IF NOT (Transfer.Mode = FIT_VFD_Transfer_Modes.Pause) AND NOT (Transfer.Mode = FIT_VFD_Transfer_Modes.Resume) THEN _w1 := Transfer.Mode; END_IF
Transfer.Config.Mode_Memory := _w1;
IF Transfer.Mode = FIT_VFD_Transfer_Modes.Resume THEN _w2 := Transfer.Config.Mode_Memory; END_IF
Transfer.Mode := _w2;
Transfer.Status := SEL(False, SEL(BCV_Not_Ready, SEL(ACV_Not_Ready, SEL(Transfer.Mode=FIT_VFD_Transfer_Modes.Lock_Out, SEL(False, SEL(Complete, SEL(Transfer_Running, SEL(FIT.PLC_Reset, SEL(IDLE_Return, SEL(PAUSED, Transfer_status.IDLE, Transfer_status.Paused), Transfer_status.IDLE), Transfer_status.FIT_Reset), Transfer_status.Running), Transfer_status.Complete), Transfer_status.Complete), Transfer_status.LOCKED_OUT), Transfer_status.ACV_Not_Ready), Transfer_status.BCV_Not_Ready), Transfer_status.VFD_Not_Ready);
_w3 := Transfer.Mode = FIT_VFD_Transfer_Modes.Idle;
_w4 := True AND NOT (ACV.Mode = ACV_Modes.Auto);
ACV_Not_Ready := _w3 AND _w4;
_w5 := _w4 OR False;
SR2(SET1 := _w3 AND _w5, RESET := NOT _w5); // SR
IF SR2.Q1 THEN _w6 := FIT_VFD_Transfer_Modes.Idle; END_IF
Transfer.Mode := _w6;
_w7 := Transfer.Status = Transfer_Status.Complete;
_w8 := Transfer_Status.IDLE = Transfer.Status OR False OR Transfer.Status = Transfer_Status.LOCKED_OUT;
_w9 := Transfer.Status = Transfer_Status.BCV_Not_Ready;
_w10 := Transfer.Mode = FIT_VFD_Transfer_Modes.Pause;
PAUSED := _w10;
_w11 := Transfer.Mode = FIT_VFD_Transfer_Modes.IDLE;
_w12 := Complete OR Error OR _w11 OR _w10;
CTRL_PID_1(
    ACT := FIT.Rate,
    SET := Transfer.Config.Target_Rate,
    SUP := 0.0,
    OFS := Transfer.Config.Target_Rate * Transfer.Config.FF,
    M_I := 0.0,
    MAN := _w12,
    RST := _w12,
    KP := Transfer.Config.KP,
    TN := Transfer.Config.TN,
    TV := Transfer.Config.TV,
    LL := 0,
    LH := 100); // BURKERT_OSCAT_BASIC.CTRL_PID
PID_CV := CTRL_PID_1.Y;
TP11(IN := NOT LockOut_Active AND _w12, PT := t#2s); // TP
ACV.PLC_CMD := SEL(TP11.Q, ACV.PLC_CMD, 0.0);
IDLE_Return := _w9 AND _w11;
SR_10(SET1 := FIT.Total<1, RESET := _w11); // SR
TON_10(IN := SR_10.Q1, PT := T#2s); // TON
FIT_Reset_Complete := TON_10.Q;
R_TRIG_0(CLK := _w11 OR TON_10.Q); // R_trig
_w13 := SEL(R_TRIG_0.Q, FIT.PLC_Reset, False);
_w14 := Transfer.Mode = FIT_VFD_Transfer_Modes.Batch;
_w15 := _w14 AND FIT_Reset_Complete AND FIT.Total >= Transfer.Config.Target_Volume;
Batch_Complete := _w15;
RS_11(SET := Time_Complete OR _w15 OR False, RESET1 := _w11); // RS
Complete := RS_11.Q1;
_w16 := LOCK_OUT AND _w8 AND NOT RS_11.Q1;
F_TRIG_10(CLK := _w16); // F_Trig
IF F_TRIG_10.Q THEN _w17 := FIT_VFD_Transfer_Modes.Idle; END_IF
Transfer.Mode := _w17;
_w18 := _w16;
IF _w18 THEN _w19 := FIT_VFD_Transfer_Modes.Lock_Out; END_IF
LockOut_Active := _w18;
Transfer.Mode := _w19;
FIT.PLC_Reset := SEL(NOT SR_10.Q1 AND _w14 AND NOT _w15, _w13, True);
_w20 := _w14 AND FIT_Reset_Complete AND NOT Complete AND NOT Error AND NOT Time_Complete;
Transfer_Running := _w20;
transfer.Remaining_Volume := SEL(_w20, Transfer.Config.Target_Volume, Transfer.Config.Target_Volume-fit.Total);
ACV.PLC_CMD := SEL(_w20, ACV.PLC_CMD, PID_CV);
TON_12(IN := _w7, PT := T#10s); // TON

END_FUNCTION_BLOCK

// 20 Program Organization Units/Level_2_Controls/Batch
FUNCTION_BLOCK Batch
VAR_INPUT
	Rate_PID: REFERENCE TO PID_Control;
	Config:	REFERENCE TO cBatch;
	FIT_Total:REAL;
	FIT_Rate:REAL;
	
END_VAR
VAR_OUTPUT
	FIT_Reset:BOOL;
END_VAR
VAR
	Local_Status:eBatch_Status;
	Local_task:eBatch_Task;
	Local_mode:eHOA_Modes;
	
	Start_Rate:REAL;
	End_Rate:REAL;
	
END_VAR

//AUX(); Now Called From Methods


CASE Config.Line_Mode.eMode OF
	eHOA_Modes.Auto:Mode_Auto();
	eHOA_Modes.Manual:Mode_Manual();
	eHOA_Modes.Off:Mode_OFF();
	
END_CASE;

CASE Config.Line_Task.eTask OF
	eBatch_Task.OFF:Task_off();
	eBAtch_Task.Pause:Task_Pause();
	eBatch_Task.Resume:Task_Resume();
	eBatch_task.Run:Task_Run();
	
END_CASE

END_FUNCTION_BLOCK

// 20 Program Organization Units/Transfer_ACV_VFD_FIT_UDFB
FUNCTION_BLOCK Transfer_ACV_VFD_FIT_UDFB
VAR_INPUT
	//Index:INT;
	LOCK_OUT:BOOL:=FALSE;
	
END_VAR
VAR_OUTPUT
END_VAR
VAR
	Paused:BOOL;
	Idle_return:BOOL;
	Transfer_Running:BOOL;
	Complete:BOOL;
	ACV_Not_Ready:BOOL;
	VFD_Not_Ready:BOOL;
	BCV_Not_Ready:BOOL;
	Time_Complete:BOOL;
	FIT_Reset_Complete:BOOL;
	Pump_Start:BOOL;
	Lockout_Active:BOOL;
	Error:BOOL;
	Flow_Mode:BOOL;
	Batch_Complete:BOOL;
	Enable_pump:BOOL;
	
	PID_CV:REAL;
	
	
	
	
	SR2: SR;
	TON_0: TON;
	CTRL_PID_1: BURKERT_OSCAT_BASIC.CTRL_PID;
	R_TRIG_0: R_trig;
	TON_10: TON;
	SR_10: SR;
	RS_11: RS;
	TON_12: TON;
	F_TRIG_10: F_Trig;
	TP11: TP;
END_VAR

VAR_IN_OUT
	Transfer:FIT_VFD_Transfer_DUT;
	VFD:VFD_Vacon_DUT;
	ACV:ACV_DUT;
	FIT:FIT_DUT;
	
END_VAR
VAR // added by the converter: edge detectors and wires of the graphical bodies
    _w1, _w2, _w7, _w22, _w24 : ANY;
    _w3, _w4, _w5, _w6, _w8, _w9, _w10, _w11, _w12, _w13, _w14, _w15, _w16, _w17, _w18, _w19, _w20, _w21, _w23, _w25 : BOOL;
END_VAR

IF NOT (Transfer.Mode = FIT_VFD_Transfer_Modes.Pause) AND NOT (Transfer.Mode = FIT_VFD_Transfer_Modes.Resume) THEN _w1 := Transfer.Mode; END_IF
Transfer.Config.Mode_Memory := _w1;
IF Transfer.Mode = FIT_VFD_Transfer_Modes.Resume THEN _w2 := Transfer.Config.Mode_Memory; END_IF
Transfer.Mode := _w2;
Transfer.Status := SEL(VFD_Not_Ready, SEL(BCV_Not_Ready, SEL(ACV_Not_Ready, SEL(Transfer.Mode=FIT_VFD_Transfer_Modes.Lock_Out, SEL(False, SEL(Complete, SEL(Transfer_Running, SEL(FIT.PLC_Reset, SEL(IDLE_Return, SEL(PAUSED, Transfer_status.IDLE, Transfer_status.Paused), Transfer_status.IDLE), Transfer_status.FIT_Reset), Transfer_status.Running), Transfer_status.Complete), Transfer_status.Complete), Transfer_status.LOCKED_OUT), Transfer_status.ACV_Not_Ready), Transfer_status.BCV_Not_Ready), Transfer_status.VFD_Not_Ready);
_w3 := Transfer.Mode = FIT_VFD_Transfer_Modes.Idle;
_w4 := True AND NOT (ACV.Mode = ACV_Modes.Auto);
ACV_Not_Ready := _w3 AND _w4;
_w5 := True AND NOT (VFD.CONTROL.MODE = VFD_Modes.Auto);
_w6 := _w4 OR _w5;
SR2(SET1 := _w3 AND _w6, RESET := NOT _w6); // SR
IF SR2.Q1 THEN _w7 := FIT_VFD_Transfer_Modes.Idle; END_IF
Transfer.Mode := _w7;
VFD_Not_Ready := _w3 AND _w5;
_w8 := Transfer.Status = Transfer_Status.Complete;
_w9 := Transfer.Status = Transfer_Status.BCV_Not_Ready OR Transfer.Status = Transfer_Status.VFD_Not_Ready;
_w10 := Transfer_Status.IDLE = Transfer.Status OR False OR Transfer.Status = Transfer_Status.LOCKED_OUT;
_w11 := Transfer.Mode = FIT_VFD_Transfer_Modes.Pause;
PAUSED := _w11;
_w12 := Transfer.Mode = FIT_VFD_Transfer_Modes.IDLE;
_w13 := Complete OR Error OR _w12 OR _w11;
_w14 := NOT Pump_Start OR _w13;
CTRL_PID_1(
    ACT := FIT.Rate,
    SET := Transfer.Config.Target_Rate,
    SUP := 0.0,
    OFS := Transfer.Config.Target_Rate * Transfer.Config.FF,
    M_I := 0.0,
    MAN := _w14,
    RST := _w14,
    KP := Transfer.Config.KP,
    TN := Transfer.Config.TN,
    TV := Transfer.Config.TV,
    LL := 0,
    LH := 100); // BURKERT_OSCAT_BASIC.CTRL_PID
PID_CV := CTRL_PID_1.Y;
TP11(IN := NOT LockOut_Active AND _w13, PT := t#2s); // TP
VFD.CONTROL.PLC_Run := SEL(TP11.Q, VFD.CONTROL.PLC_Run, FALSE);
VFD.CONTROL.PLC_CMD := SEL(TP11.Q, VFD.CONTROL.PLC_CMD, 0.0);
ACV.PLC_CMD := SEL(TP11.Q, ACV.PLC_CMD, 0.0);
IDLE_Return := _w9 AND _w12;
SR_10(SET1 := FIT.Total<1, RESET := _w12); // SR
TON_10(IN := SR_10.Q1, PT := T#2s); // TON
FIT_Reset_Complete := TON_10.Q;
R_TRIG_0(CLK := _w12 OR TON_10.Q); // R_trig
_w15 := SEL(R_TRIG_0.Q, FIT.PLC_Reset, False);
_w16 := Transfer.Mode = FIT_VFD_Transfer_Modes.Batch;
_w17 := False OR False OR _w16;
Flow_Mode := _w17;
_w18 := _w17 AND FIT_Reset_Complete AND NOT Complete AND NOT Error AND NOT Time_Complete;
Transfer_Running := _w18;
transfer.Remaining_Volume := SEL(_w18, Transfer.Config.Target_Volume, Transfer.Config.Target_Volume-fit.Total);
_w19 := True AND _w18;
Enable_Pump := _w19;
ACV.PLC_CMD := SEL(_w19, ACV.PLC_CMD, PID_CV);
_w20 := _w16 AND FIT_Reset_Complete AND FIT.Total >= Transfer.Config.Target_Volume;
Batch_Complete := _w20;
RS_11(SET := Time_Complete OR _w20 OR False, RESET1 := _w12); // RS
Complete := RS_11.Q1;
_w21 := LOCK_OUT AND _w10 AND NOT RS_11.Q1;
F_TRIG_10(CLK := _w21); // F_Trig
IF F_TRIG_10.Q THEN _w22 := FIT_VFD_Transfer_Modes.Idle; END_IF
Transfer.Mode := _w22;
_w23 := _w21;
IF _w23 THEN _w24 := FIT_VFD_Transfer_Modes.Lock_Out; END_IF
LockOut_Active := _w23;
Transfer.Mode := _w24;
FIT.PLC_Reset := SEL(NOT SR_10.Q1 AND _w17 AND NOT _w20, _w15, True);
_w25 := SEL(_w19, _w18, ACV.Valve_Actual >= 5);
Pump_Start := _w25;
VFD.CONTROL.PLC_CMD := SEL(_w25, VFD.CONTROL.PLC_CMD, PID_CV);
VFD.CONTROL.PLC_Run := SEL(_w25, VFD.CONTROL.PLC_Run, PID_CV > 15);
TON_12(IN := _w8, PT := T#10s); // TON

END_FUNCTION_BLOCK

// 20 Program Organization Units/Transfer_BCV_FIT_UDFB
FUNCTION_BLOCK Transfer_BCV_FIT_UDFB
VAR_INPUT
	LOCK_OUT:BOOL:=FALSE;
	//FIT_Rate:REAL;
	//FIT_Volume:REAL;
	//Valve_Ready:BOOL;
	
END_VAR
VAR_OUTPUT
	//BCV:BOOL;
	//ACV:REAL:
END_VAR
VAR
	Paused:BOOL;
	Idle_return:BOOL;
	Transfer_Running:BOOL;
	Complete:BOOL;
	ACV_Not_Ready:BOOL;
	//VFD_Not_Ready:BOOL;
	BCV_Not_Ready:BOOL;
	Time_Complete:BOOL;
	FIT_Reset_Complete:BOOL;
	//Pump_Start:BOOL;
	Lockout_Active:BOOL;
	Error:BOOL;
	Flow_Mode:BOOL;
	Batch_Complete:BOOL;
	Enable_pump:BOOL;
	
	//PID_CV:REAL;
	
	
	
	
	SR2: SR;
	TON_0: TON;
	CTRL_PID_1: BURKERT_OSCAT_BASIC.CTRL_PID;
	R_TRIG_0: R_trig;
	TON_10: TON;
	SR_10: SR;
	RS_11: RS;
	TON_12: TON;
	F_TRIG_10: F_Trig;
	TP11: TP;
	FT_PIDW_1: BURKERT_OSCAT_BASIC.FT_PIDW;
	F_TRIG_0: F_Trig;
END_VAR

VAR_IN_OUT
	Transfer:FIT_Transfer_DUT;
	//FIT_Reset:BOOL;
	//VFD:VFD_Vacon_DUT;
	BCV:BCV_DUT;
	FIT:FIT_DUT;
	
END_VAR
VAR // added by the converter: edge detectors and wires of the graphical bodies
    _w1, _w2, _w5, _w6, _w20, _w22, _w23 : ANY;
    _w3, _w4, _w7, _w8, _w9, _w10, _w11, _w12, _w13, _w14, _w15, _w16, _w17, _w18, _w19, _w21 : BOOL;
END_VAR

